PROGRAM MAIN
VAR
	arrInputs		AT %I* : ARRAY[0..7] OF BOOL;
	arrOutputs		AT %Q* : ARRAY[0..7] OF BOOL;
	
	manualMap		AT %I* : INT;
	
	axisRef			: AXIS_REF;
END_VAR

END_PROGRAM

(* stored: Version 1.1.0.1
   POU MAIN: Id {a16db61f-33d9-4e15-aec8-66b56be237dc}, SpecialFunc None *)
